KUKA KRL data list: MIPO.dat

&ACCESS RVO1
DEFDAT MIPO PUBLIC
DECL REAL BOUND = -999
ENDDAT
